TYPE ST_WXT530 :
STRUCT
	stWindData			:ST_WindData;
END_STRUCT
END_TYPE

(* stored: Version 1.1.0.1, ProductVersion 3.1.4020.6
   DUT ST_WXT530: Id {d4d8c47d-2322-4eb0-b15f-97b95463dc5e} *)
